FUNCTION_BLOCK BLOCK_POMP_1E_PCR_PPM_ASS_ETHERCAT

(* Historique des versions*)
(* VERSION 1.0 - 05/2015 - GV - affaire 9070*)
(* VERSION 2.0 - 10/2022 - GV - ajout gestion roots *)


(* BLOCK GESTION POMPAGE CRYO ON BOARD ENCEINTE *)
(*	Gestion pompage enceinte sans sas constitué de :
	Pompe primaire pour prévidage, regen cryo et pompage interjoint
	Pompe cryogénique on-board CTI pour le pompage secondaire
	Vanne de pompage primaire enceinte
	Vanne de remise à atmosphère enceinte
	Vanne de pompage inter-joint (optionnelle)
	Vanne secondaire asservie, pilotée par ethercatf
*)

VAR_INPUT
(*information générale*)
	RESET:					BOOL;
	MANUAL:					BOOL;
	CTRL_PLC:				BOOL;
	I_Prep_Ventil_Ok:		BOOL;		(*information externe indiquant que l'enceinte est prête à être ventilée par ex. circulation d'eau à l'arrêt
										ou polycold arreté ou basculement en eau chaude ok ...*)
	I_Fin_Ventil:			BOOL;		(*information externe de fin de ventilation de l'enceinte  *)
	I_Stop_Mesure_OK:		BOOL;		(*information externe indiquant que les jauges ont été stoppées prélablement à la ventilation de l'enceinte*)
	IN_Pressure_RP:			REAL;		(*interfaçage avec M11.state_pression du PRG correspondant*)
	I_Ref_OK:				BOOL;		(*information externe indiquant que le refroidissement est ok pour démarrer les pompes*)
	
(*Gestion régen partielle*)
	IN_Temp_Etage1:			REAL;
	PRM_Temp_Post_Purge:	REAL;
	PRM_Tim_Post_Purge:		TIME;

(*Paramètres et commandes du test de remontée de pression*)
	PRM_Pr_test:			REAL;		(*Pression initiale de test de remontée*)
	PRM_Tim_test:			TIME;		(*Durée d'attente en test*)
	CO_Stop_Test_RP:		BOOL;		(*Demande arrêt test remontée de pression*)

(*sécurité*)
	IN_FE11T:				BOOL;		(*indicateur enceinte fermée - capteur 1*)
	IN_FE12T:				BOOL;		(*indicateur enceinte fermée - capteur 2*)
	IN_VT11F:				BOOL;		(*clapet SAS enceinte fermé*)

(*seuil de vide*)
	TH_Vide_Primaire:		BOOL;		(*Pression enceinte <= Seuil de fin de pompage primaire*)
	TH_Grosse_Fuite:		BOOL;		(*Pression enceinte <= Seuil de detection de grosse fuite enceinte*)
	TH_Atm:					BOOL;		(*pression enceinte >= Seuil pression atm. de fin de ventilation*)
	TH_RP_Enc:				BOOL;		(*pression enceinte <= Pression max. dans l'enceinte*)
	TH_Test_RP:				BOOL;		(*Pression <= Seuil de pression de test*)

(*composant de la fonction*)
	VP11:					BLOCK_ACTUATOR;									(*vanne de pompage primaire enceinte *)
	VH11:					BLOCK_ACTUATOR;									(*vanne de ventilation de l'enceinte*)
	PP11:					BLOCK_PPM;										(*Pompe primaire enceinte*)
	PR11:					BLOCK_PPM;										(*Pompe roots enceinte*)
	PS11:					BLOCK_PCR_CTI_OB;								(*Pompe cryogénique on board  enceinte*)
	VS11:					BLOCK_VVAT_653_ETHERCAT;						(*Vanne secondaire asservie pompage enceinte*)
	VINT:					BLOCK_ACTUATOR;									(*Vanne de pompage dans les interjoints*)

(*défaut*)
	DEF_PPrim:				PRCDEF;										(*défaut temps de pompage primaire dans l'enceinte*)
	DEF_Vent:				PRCDEF;										(*défaut temps de ventilation enceinte*)
	DEF_RP_enc:				PRCDEF;	 									(*défaut perte seuil de pompage primaire en pompage secondaire*)
	DEF_TGF:				PRCDEF;										(*défaut détection trés grosse fuite*)

(*opération*)
	OP_Marche_Pompes:			BLOCK_OPERATION;								(*opération marche pompe*)
	OP_Arret_Pompes:			BLOCK_OPERATION;								(*opération arrêt pompe*)
	OP_Isolement:				BLOCK_OPERATION;								(*opération stand-by*)
	OP_Ventilation:				BLOCK_OPERATION;								(*opération ventilation*)
	OP_Pompage_Sec:				BLOCK_OPERATION;								(*opération pompage secondaire*)
	OP_Pompage_Prim:			BLOCK_OPERATION;								(*opération pompage primaire*)
	OP_Pompage_Proc:			BLOCK_OPERATION;								(*opération pompage en procédé*)
	OP_Purge:					BLOCK_OPERATION;								(*opération purge*)
	OP_Regen:					BLOCK_OPERATION;								(*opération régénération pompe cryogénique*)
	OP_Regen_Part:				BLOCK_OPERATION;								(*opération de régénération partielle pompe cryogénique*)
	OP_Test_RP:					BLOCK_OPERATION;								(*opération test RP*)
	G7_pompage_interjoint:		BLOCK_G7;

END_VAR

VAR_INPUT PERSISTENT
(*paramètre*)
	PRM_Tim_SurVentil_E:		TIME;	(*durée du temps de surventilation*)
	PRM_Tim_Purge:				TIME;	(*durée du maintien pompage primaire en purge*)
	PRM_Tim_Arret_PP11:			TIME;	(*durée avant arrêt de la pompe primaire*)
	PRM_Pr_Atm:					REAL;	(*Pression atmosphérique dans l'enceinte*)
	PRM_Pr_PPrim:				REAL;	(*Pression de fin de pompage primaire dans l'enceinte*)
	PRM_Pr_RP_PPrim:			REAL;	(*Pression max admissible dans l'enceinte en pompage secondaire dans l'enceinte*)
	PRM_Pr_TGF:					REAL;	(*Pression de détection trés grosse fuite dans l'enceinte*)
	PRM_N_Purge:				USINT;	(*Nombre de cycles de purge pompage/ventilation*)
	CONF_Pompage_interjoint:	BOOL;	(*Utilisation de la pompe primaire pour le pompage interjoint sur l'enceinte*)
	CONF_VINT:					BOOL;	(*Utilisation d'une vanne d'isolement sur le pompage interjoint*)
	CONF_Volume_Enceinte:		REAL;	(*Volume pour RP*)

	PRM_Tim_Prep_Ventil:		TIME;	(*temporisation de prép ventilation (eau chaude suffisemment longtemps) *)

	(*Entité*)
	IsAssembly:		BOOL;		(*entité : ensemble*)
	IdXML:			STRING;		(*nom entité : identifiant pour recherche dans dico*)
	TagXML:			UINT;		(*nom entité : identifiant pour recherche dans dico*)
	IdParent:		STRING;		(*MNEMO de l'appelant*)
	MNEMO:			STRING;		(*MNEMO de l'entité*)
END_VAR


VAR_OUTPUT
	RQ_Prep_Ventil_Enc:		BOOL;											(*demande de préparation avant ventilation (réchauffement, arrêt eau ....*)
	RQ_Stop_Mesure_Enc:		BOOL;											(*demande d'arrêt de la mesure avant ventilation - Les blocs jauges concernés utilise
																			cette information pour stoppée les jauges préalablement à la ventilation*)
END_VAR

VAR_IN_OUT
END_VAR

VAR
	VAR_Reset_Sortie:					BOOL;
	TIMER_SurVentilation_Enc:			TON;		(*Temporistion de surventilation enceinte*)
	TIMER_Purge:						TON;		(*Temporisation de maintien pompage primaire en purge*)
	TIMER_Pompage_Interjoint:			TON;		(*Temporisation d'ouverture de la vanne de pompage interjoint*)
	TIMER_Arret_Roots:					TON;		(*Temporisation arrêt roots après prévidage*)
	TIMER_Arret_PP11:					TON;		(*Temporisation arrêt pompe primaire*)
	VAR_mem_isolement:					BOOL;
	VAR_Iter_Purge:						USINT;

	(*Pour RP*)
	VAR_Mem_Pression_Deb:		REAL;
	VAR_Mem_Pression_Fin:		REAL;
	VAR_Indicateur_Test:		REAL; 		(*résultat final*)
	TIMER_attente_test:			TON;		(*Temporisation pour test de remontée en pression*)
	FM_etape4:					R_TRIG;

	(*Pour prep ventil*)
	TIM_Prep_ventil:			TON;		(*timer de préparation ventil*)

	(*Pour regen*)
	FM_REGEN:						R_TRIG;		(* FM pompe cryogénique en régénération*)
	FD_REGEN:						F_TRIG;		(* FD pompe cryogénique en régénération*)
	TIMER_Post_Purge:				TON;		(*tempo max attente de retombée température après purge en regen partielle*)
	TIMER_etape6_regen:				TON;
END_VAR

PRL();

(*appel des opérations*)
ACT_ARRET_POMPES();
ACT_ISOLEMENT();
ACT_MARCHE_POMPES();
ACT_POMPAGE_PRIM();
ACT_POMPAGE_PROC();
ACT_POMPAGE_SEC();
ACT_VENTILATION();
ACT_PURGE();
ACT_REGEN();
ACT_REGEN_PART();
ACT_TEST_RP();
ACT_POMPAGE_INTERJOINT();

(*action en sortie*)
POST();

ACTION ACT_ARRET_POMPES:
(* OPERATION ARRET POMPES*)
(* arrêt des pompes*)

(*initialisation de l'opération*)
OP_ARRET_POMPES(
	CTRL_PLC:= CTRL_PLC,
	RESET:= RESET,
	ENABLE_INT:=TRUE,
	MANUAL:= MANUAL,
	ON_AUTO_INT:= (PP11.STATE_NOK AND PR11.STATE_NOK) AND (NOT OP_Pompage_Prim.Etape.0 OR NOT OP_Purge.Etape.0),
	RESTART_ENABLE_IF_OK:= FALSE,
	N_STEP_OP_OK:= 5,
	N_STEP_OP_NOK:=0);

(*appel de l'action de préparation de l'opération*)
OP_ARRET_POMPES.PRL();


(*GRAFCET*)
(* initialisation du grafcet*)
IF 		OP_Arret_Pompes.ETAPE = 0 THEN
				OP_Arret_Pompes.ETAPE.0 := TRUE;
(*repositionnement sur étape 0*)
ELSIF	MANUAL OR RESET OR OP_Marche_Pompes.ETAPE.1 THEN
				OP_Arret_Pompes.ETAPE := 0;			(*RAZ grafcet*)
				OP_Arret_Pompes.ETAPE.0:=TRUE;
(*étape 0-1*)
ELSIF 	OP_Arret_Pompes.ETAPE.0
		AND OP_Arret_Pompes.MARCHE_OP THEN
				OP_Arret_Pompes.ETAPE.1:=TRUE;
				OP_Arret_Pompes.ETAPE.0:=FALSE;
(*étape 1-2*)
ELSIF	OP_Arret_Pompes.ETAPE.1
		AND OP_Marche_Pompes.ETAPE.0  THEN
				OP_Arret_Pompes.Etape.2:=TRUE;
				OP_Arret_Pompes.Etape.1:=FALSE;
(*étape 2-3*)
ELSIF 	OP_Arret_Pompes.Etape.2
		AND (OP_Isolement.OK OR VAR_mem_isolement)
		AND (VINT.STATE_Off OR NOT CONF_VINT)
		 THEN
				OP_Arret_Pompes.Etape.3:=TRUE;
				OP_Arret_Pompes.Etape.2:=FALSE;
(*étape 3-4*)
ELSIF 	OP_Arret_Pompes.Etape.3
		AND	Timer_Arret_PP11.Q THEN 
				OP_Arret_Pompes.Etape.4:=TRUE;
				OP_Arret_Pompes.Etape.3:=FALSE;
(*étape 4-5*)
ELSIF	OP_Arret_Pompes.Etape.4
		AND PP11.STATE_Off AND PR11.STATE_Off AND PS11.STATE_Ar THEN
				OP_Arret_Pompes.Etape.5:=TRUE;
				OP_Arret_Pompes.Etape.4:=FALSE;
END_IF;

(*cloture du traitement de l'opération*)
OP_Arret_Pompes.POST();

(************************************************************************)
(*Gestion de la mémoire de la demande d'isolement de l'enceinte*)
(************************************************************************)
IF 		OP_Ventilation.Etape.9 THEN
	VAR_mem_isolement	:=	TRUE;
ELSIF	NOT OP_Pompage_Prim.AR OR NOT OP_Pompage_Sec.AR OR NOT OP_Pompage_Proc.AR OR NOT OP_Purge.AR THEN
	VAR_mem_isolement	:=	FALSE;
END_IF
(*IF OP_Arret_pompes.Etape.2 AND (NOT OP_Pompage_Prim.Etape.0  OR NOT OP_Pompage_Proc.Etape.0 OR NOT OP_Pompage_Sec.Etape.0) THEN
	VAR_mem_isolement_enceinte := TRUE;
END_IF;
IF OP_Arret_pompes.Etape.0 OR OP_Arret_Pompes.Etape.3 THEN
	VAR_mem_isolement_enceinte := FALSE;
END_IF;*)
END_ACTION

ACTION ACT_ISOLEMENT:
(*OPERATION ISOLEMENT ENCEINTE*)
(*isolement de l'enceinte*)

(*initialisation de l'opération*)
OP_Isolement(
	CTRL_PLC:= CTRL_PLC,
	RESET:= RESET,
	ENABLE_INT:=TRUE,
	MANUAL:= MANUAL,
	ON_AUTO_INT:= 	((DEF_TGF.DEF OR DEF_RP_enc.DEF) AND (NOT OP_Pompage_Prim.Etape.0 OR NOT OP_Pompage_Sec.Etape.0 OR NOT OP_Pompage_proc.Etape.0))
					OR (PS11.STATE_Nok AND (NOT OP_Pompage_Sec.Etape.0 OR NOT OP_Pompage_proc.Etape.0))
					OR (PP11.STATE_Nok AND NOT OP_Pompage_Prim.Etape.0)
					OR (PR11.STATE_NOK AND NOT OP_Pompage_Prim.Etape.0),
	RESTART_ENABLE_IF_OK:= FALSE,
	N_STEP_OP_OK:= 4,
	N_STEP_OP_NOK:=0);

(*appel de l'action de préparation de l'opération*)
OP_Isolement.PRL();


(*GRAFCET*)
(* initialisation du grafcet*)
IF 		OP_Isolement.Etape = 0
		THEN
				OP_Isolement.Etape.0	:= TRUE;
(*repositionnement sur étape 0*)
ELSIF	MANUAL OR RESET OR OP_pompage_sec.Etape.1 OR OP_Pompage_Proc.Etape.1 OR Op_Pompage_Prim.Etape.1
		OR OP_ventilation.Etape.2 OR OP_Ventilation.Etape.9 OR OP_Purge.Etape.1 THEN
				OP_Isolement.Etape := 0;
				OP_Isolement.Etape.0:=TRUE;
(*étape 0-1*)
ELSIF 	OP_Isolement.Etape.0
		AND(
		OP_Isolement.Marche_OP OR
		OP_ventilation.Etape.1 OR
		OP_Test_RP.Etape.3 OR
		(OP_Arret_Pompes.Etape.2 AND NOT VAR_mem_isolement) OR
		OP_Regen.Etape.2 OR OP_Regen_Part.Etape.2
		)
		THEN
				OP_Isolement.Etape.1:=TRUE;
				OP_Isolement.Etape.0:=FALSE;
(*étape 1-2*)
ELSIF	OP_Isolement.Etape.1
		AND OP_Pompage_Proc.Etape.0
		AND OP_Pompage_Prim.Etape.0
		AND OP_Pompage_Sec.Etape.0
		AND (OP_Ventilation.Etape.0 OR OP_Ventilation.Etape.1)
		AND (OP_Purge.Etape.0 OR (OP_Purge.Etape.4 AND OP_Ventilation.Etape.1))
		THEN
				OP_Isolement.Etape.2:=TRUE;
				OP_Isolement.Etape.1:=FALSE;
(*étape 2-3*)
ELSIF 	OP_Isolement.Etape.2 AND
		VP11.STATE_Off AND
		VS11.STATE_Off AND
		VH11.STATE_Off  THEN
				OP_Isolement.Etape.3:=TRUE;
				OP_Isolement.Etape.2:=FALSE;
(*étape 3-4*)
ELSIF	OP_Isolement.Etape.3
		AND ((PP11.STATE_Off AND PR11.STATE_Off) OR PS11.STATE_Regen OR CONF_Pompage_interjoint) THEN
				OP_isolement.Etape.4:=TRUE;
				OP_isolement.Etape.3:=FALSE;
END_IF;

(*cloture du traitement de l'opération*)
OP_Isolement.POST();
END_ACTION

ACTION ACT_MARCHE_POMPES:
(* OPERATION MARCHE POMPES*)
(* mise en marche des pompes*)

(*initialisation de l'opération*)
OP_MARCHE_POMPES(
	CTRL_PLC:= CTRL_PLC,
	RESET:= RESET,
	ENABLE_INT:=TRUE,
	MANUAL:= MANUAL,
	ON_AUTO_INT:= TRUE,
	RESTART_ENABLE_IF_OK:= FALSE,
	N_STEP_OP_OK:= 5,
	N_STEP_OP_NOK:=0);

(*appel de l'action de préparation de l'opération*)
OP_MARCHE_POMPES.PRL();


(*GRAFCET*)
(* initialisation du grafcet*)
IF 		OP_MARCHE_POMPES.ETAPE = 0
		THEN
				OP_MARCHE_POMPES.ETAPE.0 := TRUE;
(*repositionnement sur étape 0*)
ELSIF	MANUAL OR RESET OR OP_ARRET_POMPES.ETAPE.1
		THEN
				OP_MARCHE_POMPES.ETAPE := 0;			(*RAZ grafcet*)
				OP_MARCHE_POMPES.ETAPE.0:=TRUE;
(*étape 0-1*)
ELSIF 	OP_MARCHE_POMPES.ETAPE.0
		AND (OP_MARCHE_POMPES.MARCHE_OP OR OP_POMPAGE_SEC.ETAPE.2
			OR (OP_Regen.Etape.5 AND TH_Atm))
		THEN
				OP_MARCHE_POMPES.ETAPE.1:=TRUE;
				OP_MARCHE_POMPES.ETAPE.0:=FALSE;
(*étape 1-2*)
ELSIF	OP_MARCHE_POMPES.ETAPE.1
		AND OP_ARRET_POMPES.ETAPE.0 AND PR11.STATE_Off AND I_Ref_Ok
		THEN
				OP_MARCHE_POMPES.ETAPE.2:=TRUE;
				OP_MARCHE_POMPES.ETAPE.1:=FALSE;
(*étape 2-3*)
ELSIF 	OP_MARCHE_POMPES.ETAPE.2
		AND (PP11.STATE_On OR NOT CONF_Pompage_interjoint)
		THEN
				OP_MARCHE_POMPES.ETAPE.3:=TRUE;
				OP_MARCHE_POMPES.ETAPE.2:=FALSE;
(*étape 3-4*)
ELSIF	OP_MARCHE_POMPES.ETAPE.3
		THEN
				OP_MARCHE_POMPES.ETAPE.4:=TRUE;
				OP_MARCHE_POMPES.ETAPE.3:=FALSE;
(*étape 4-5*)
ELSIF 	OP_MARCHE_POMPES.ETAPE.4
		AND PS11.STATE_On AND PS11.STATE_Ok AND NOT PS11.STATE_Regen
		THEN
				OP_MARCHE_POMPES.ETAPE.5:=TRUE;
				OP_MARCHE_POMPES.ETAPE.4:=FALSE;
(*étape 5-4*)
ELSIF 	OP_MARCHE_POMPES.ETAPE.5
		AND (PS11.STATE_Regen OR NOT PS11.STATE_Ok)		THEN
				OP_MARCHE_POMPES.ETAPE.4:=TRUE;
				OP_MARCHE_POMPES.ETAPE.5:=FALSE;
END_IF;

(*cloture du traitement de l'opération*)
OP_MARCHE_POMPES.POST();
END_ACTION

ACTION ACT_POMPAGE_INTERJOINT:
(*GRAFCET*)
(* initialisation du grafcet*)
IF 		G7_pompage_interjoint.etape = 0
		THEN
				G7_pompage_interjoint.etape.0 := TRUE;
(*repositionnement sur étape 0*)
ELSIF	MANUAL OR RESET
		OR (NOT OP_POMPAGE_SEC.OK AND NOT OP_Pompage_Proc.OK AND NOT OP_Pompage_Proc.EC)
		OR NOT CONF_Pompage_interjoint OR NOT CONF_VINT
		THEN
				G7_pompage_interjoint.etape := 0;			(*RAZ grafcet*)
				G7_pompage_interjoint.etape.0:=TRUE;
(*étape 0-1*)
ELSIF 	G7_pompage_interjoint.etape.0
		AND (OP_POMPAGE_SEC.OK OR OP_Pompage_Proc.EC OR OP_Pompage_Proc.OK)
		THEN
				G7_pompage_interjoint.etape.1:=TRUE;
				G7_pompage_interjoint.etape.0:=FALSE;
(*étape 1-2*)
ELSIF	G7_pompage_interjoint.etape.1
		AND TIMER_pompage_interjoint.Q
		THEN
				G7_pompage_interjoint.etape.2:=TRUE;
				G7_pompage_interjoint.etape.1:=FALSE;
END_IF;

G7_pompage_interjoint.POST();
END_ACTION

ACTION ACT_POMPAGE_PRIM:
(*OPERATION POMPAGE PRIMAIRE ENCEINTE*)
(*pompage primaire dans l'enceinte*)

(*initialisation de l'opération*)
OP_POMPAGE_PRIM(
	CTRL_PLC:= CTRL_PLC,
	RESET:= RESET,
	ENABLE_INT:= OP_Purge.Etape.0 AND IN_FE11T AND IN_FE12T,
	MANUAL:= MANUAL,
	RESTART_ENABLE_IF_OK:= FALSE,
	N_STEP_OP_OK:= 5,
	N_STEP_OP_NOK:=0);

(*appel de l'action de préparation de l'opération*)
OP_POMPAGE_PRIM.PRL();


(*GRAFCET*)
(* initialisation du grafcet*)
IF 		OP_Pompage_Prim.Etape = 0
		THEN
				OP_Pompage_Prim.Etape.0:= TRUE;
(*repositionnement sur étape 0*)
ELSIF	MANUAL OR RESET OR OP_Isolement.Etape.1 OR OP_Pompage_Sec.Etape.4
		OR OP_Pompage_Proc.Etape.1
		THEN
				OP_Pompage_Prim.ETAPE := 0;
				OP_Pompage_Prim.Etape.0:=TRUE;
(*étape 0-1*)
ELSIF 	OP_Pompage_Prim.Etape.0
		AND (OP_Pompage_Prim.Marche_OP OR OP_Pompage_Sec.Etape.3 OR OP_Purge.Etape.2)
		THEN
				OP_Pompage_Prim.Etape.1:=TRUE;
				OP_Pompage_Prim.Etape.0:=FALSE;
(*étape 1-2*)
ELSIF	OP_Pompage_Prim.Etape.1
		AND OP_Isolement.Etape.0
		AND OP_Ventilation.Etape.0
		AND OP_Pompage_Proc.Etape.0
		AND (OP_Pompage_Sec.Etape.0 OR OP_Pompage_Sec.Etape.3)
		AND (OP_Purge.Etape.0 OR OP_Purge.Etape.6 OR OP_Purge.Etape.2)
		AND VS11.STATE_Off
		AND VH11.STATE_Off
		THEN
				OP_Pompage_Prim.Etape.2:=TRUE;
				OP_Pompage_Prim.Etape.1:=FALSE;

(*étape 2-3*)
ELSIF 	OP_Pompage_prim.Etape.2
		THEN
				OP_Pompage_Prim.Etape.3:=TRUE;
				OP_Pompage_Prim.Etape.2:=FALSE;
(*étape 3-4*)
ELSIF	OP_Pompage_Prim.Etape.3
		AND PP11.STATE_On AND PR11.STATE_On THEN
				OP_Pompage_Prim.Etape.4:=TRUE;
				OP_Pompage_Prim.Etape.3:=FALSE;
(*étape 4-5*)
ELSIF 	OP_Pompage_Prim.Etape.4
		AND VP11.STATE_On
		THEN
				OP_Pompage_Prim.Etape.5:=TRUE;
				OP_Pompage_Prim.Etape.4:=FALSE;
END_IF;

(*cloture du traitement de l'opération*)
OP_Pompage_Prim.POST();
END_ACTION

ACTION ACT_POMPAGE_PROC:
(*OPERATION POMPAGE PROCEDE*)
(*pompage procede dans l'enceinte*)

(*initialisation de l'opération*)
OP_Pompage_Proc(
	CTRL_PLC:= CTRL_PLC,
	RESET:= RESET,
	ENABLE_INT:= OP_POMPAGE_SEC.OK OR OP_Pompage_Proc.OK,
	MANUAL:= MANUAL,
	RESTART_ENABLE_IF_OK:= FALSE,
	N_STEP_OP_OK:= 3,
	N_STEP_OP_NOK:=0);

(*appel de l'action de préparation de l'opération*)
OP_Pompage_Proc.PRL();


(*GRAFCET*)
(* initialisation du grafcet*)
IF 		OP_Pompage_Proc.Etape = 0
		THEN
				OP_Pompage_Proc.Etape.0:= TRUE;
(*repositionnement sur étape 0*)
ELSIF	MANUAL OR RESET OR OP_Isolement.Etape.1 OR OP_Pompage_Prim.Etape.1 OR OP_Pompage_Sec.Etape.1
		OR OP_Purge.Etape.1
		THEN
				OP_Pompage_Proc.Etape := 0;
				OP_Pompage_Proc.Etape.0:=TRUE;
(*étape 0-1*)
ELSIF 	OP_Pompage_Proc.Etape.0
		AND OP_Pompage_Proc.Marche_OP
		THEN
				OP_Pompage_Proc.Etape.1:=TRUE;
				OP_Pompage_Proc.Etape.0:=FALSE;
(*étape 1-2*)
ELSIF	OP_Pompage_Proc.Etape.1
		AND OP_Pompage_Sec.Etape.0
		THEN
				OP_Pompage_Proc.Etape.2:=TRUE;
				OP_Pompage_Proc.Etape.1:=FALSE;
(*étape 2-3*)
ELSIF 	OP_Pompage_proc.Etape.2
		AND VS11.STATE_Lam THEN
				OP_Pompage_Proc.Etape.3:=TRUE;
				OP_Pompage_Proc.Etape.2:=FALSE;
(*étape 3-2*)
ELSIF 	OP_Pompage_Proc.Etape.3
		AND OP_Pompage_Proc.Marche_OP
		THEN
				OP_Pompage_Proc.Etape.2:=TRUE;
				OP_Pompage_Proc.Etape.3:=FALSE;
END_IF;

(*cloture du traitement de l'opération*)
OP_Pompage_Proc.POST();
END_ACTION

ACTION ACT_POMPAGE_SEC:
(*OPERATION POMPAGE SECONDAIRE ENCEINTE*)
(*pompage secondaire dans l'enceinte*)

(*initialisation de l'opération*)
OP_pompage_sec(
	CTRL_PLC:= CTRL_PLC,
	RESET:= RESET,
	ENABLE_INT:=IN_FE11T AND IN_FE12T AND NOT PS11.STATE_Regen,
	MANUAL:= MANUAL,
	RESTART_ENABLE_IF_OK:= FALSE,
	N_STEP_OP_OK:= 7,
	N_STEP_OP_NOK:=0);

(*appel de l'action de préparation de l'opération*)
OP_Pompage_Sec.PRL();


(*GRAFCET*)
(* initialisation du grafcet*)
IF 		OP_Pompage_Sec.Etape = 0
		THEN
				OP_Pompage_Sec.Etape.0:= TRUE;
(*repositionnement sur étape 0*)
ELSIF	MANUAL OR RESET OR OP_Isolement.Etape.1 OR OP_Pompage_Proc.Etape.1
		OR (OP_Pompage_Prim.Etape.1 AND NOT OP_Pompage_Sec.Etape.3) OR OP_Purge.Etape.1
		THEN
				OP_Pompage_Sec.Etape := 0;
				OP_Pompage_Sec.Etape.0:=TRUE;
(*étape 0-1*)
ELSIF 	OP_Pompage_Sec.Etape.0 AND
		(OP_Pompage_Sec.Marche_OP OR OP_Purge.Etape.6 OR
			OP_Test_RP.Etape.2 OR OP_Test_RP.Etape.7
		OR (OP_Regen.Etape.5 AND NOT TH_Atm AND OP_Pompage_Sec.ENABLE_INT))
		THEN
				OP_Pompage_Sec.Etape.1:=TRUE;
				OP_Pompage_Sec.Etape.0:=FALSE;
(*étape 1-2*)
ELSIF	OP_Pompage_Sec.Etape.1
		AND OP_Isolement.Etape.0
		AND OP_Ventilation.Etape.0
		AND OP_Pompage_Proc.Etape.0
		AND (OP_Purge.Etape.0 OR OP_Purge.Etape.6)
		THEN
				OP_Pompage_Sec.Etape.2:=TRUE;
				OP_Pompage_Sec.Etape.1:=FALSE;
(*étape 2-3*)
ELSIF 	OP_Pompage_Sec.Etape.2
		AND OP_MARCHE_POMPES.ok AND NOT TH_Vide_Primaire AND VH11.STATE_Off
		THEN
				OP_Pompage_Sec.Etape.3:=TRUE;
				OP_Pompage_Sec.Etape.2:=FALSE;
(*étape 2-4*)
ELSIF 	OP_Pompage_Sec.Etape.2
		AND OP_MARCHE_POMPES.ok AND TH_Vide_Primaire AND VH11.STATE_Off
		THEN
				OP_Pompage_Sec.Etape.4:=TRUE;
				OP_Pompage_Sec.Etape.2:=FALSE;
(*étape 3-4*)
ELSIF	OP_Pompage_Sec.Etape.3
		AND	OP_POMPAGE_PRIM.ok  AND TH_Vide_Primaire
		THEN
				OP_Pompage_Sec.Etape.4:=TRUE;
				OP_Pompage_Sec.Etape.3:=FALSE;
(*étape 4-5*)
ELSIF	OP_Pompage_Sec.Etape.4
		AND VP11.STATE_Off
		AND  OP_POMPAGE_PRIM.AR   THEN
				OP_Pompage_Sec.Etape.5:=TRUE;
				OP_Pompage_Sec.Etape.4:=FALSE;
(*étape 5-6*)
ELSIF 	OP_Pompage_Sec.Etape.5
		AND (PP11.STATE_Off AND PR11.STATE_Off OR CONF_Pompage_interjoint)
		THEN
				OP_Pompage_Sec.Etape.6:=TRUE;
				OP_Pompage_Sec.Etape.5:=FALSE;
(*étape 6-7*)
ELSIF 	OP_Pompage_Sec.Etape.6
		AND VS11.STATE_On
		THEN
				OP_Pompage_Sec.Etape.7:=TRUE;
				OP_Pompage_Sec.Etape.6:=FALSE;
END_IF;

(*cloture du traitement de l'opération*)
OP_Pompage_Sec.POST();
END_ACTION

ACTION ACT_PURGE:
(*OPERATION PURGE*)
(*purge enceinte : pompage primaire pendant un temps donné puis ventilation, répété X fois*)

(*initialisation de l'opération*)
OP_Purge(
	CTRL_PLC:= CTRL_PLC,
	RESET:= RESET,
	ENABLE_INT:= IN_FE11T AND IN_FE12T AND OP_Test_RP.AR,
	MANUAL:= MANUAL,
	RESTART_ENABLE_IF_OK:= FALSE,
	N_STEP_OP_OK:= 7,
	N_STEP_OP_NOK:=0);

(*appel de l'action de préparation de l'opération*)
OP_Purge.PRL();


(*GRAFCET*)
(* initialisation du grafcet*)
IF 		OP_Purge.Etape = 0
		THEN
				OP_Purge.Etape.0:= TRUE;
(*repositionnement sur étape 0*)
ELSIF	MANUAL OR RESET OR OP_Arret_Pompes.Etape.1
		OR (OP_Isolement.Etape.1 AND NOT OP_Ventilation.Etape.1)
		OR (OP_Pompage_Sec.Etape.1 AND NOT OP_Purge.Etape.6)
		THEN
				OP_Purge.Etape := 0;
				OP_Purge.Etape.0:=TRUE;
(*étape 0-1*)
ELSIF 	OP_Purge.Etape.0
		AND OP_Purge.Marche_OP
		THEN
				OP_Purge.Etape.1:=TRUE;
				OP_Purge.Etape.0:=FALSE;
(*étape 1-2*)
ELSIF	OP_Purge.Etape.1
		AND OP_Pompage_Sec.Etape.0 AND OP_Pompage_Prim.Etape.0 AND OP_Pompage_Proc.Etape.0
		AND OP_Ventilation.Etape.0 AND OP_Isolement.Etape.0
		THEN
				OP_Purge.Etape.2:=TRUE;
				OP_Purge.Etape.1:=FALSE;
(*étape 2-3*)
ELSIF 	OP_Purge.Etape.2
		AND OP_Pompage_Prim.OK AND TH_Vide_Primaire
		THEN
				OP_Purge.Etape.3:=TRUE;
				OP_Purge.Etape.2:=FALSE;
(*étape 3-4*)
ELSIF 	OP_Purge.Etape.3
		AND TIMER_Purge.Q
		THEN
				OP_Purge.Etape.4:=TRUE;
				OP_Purge.Etape.3:=FALSE;
(*étape 3-2*)
ELSIF 	OP_Purge.Etape.3
		AND NOT OP_Pompage_Prim.OK
		THEN
				OP_Purge.Etape.2:=TRUE;
				OP_Purge.Etape.3:=FALSE;
(*étape 4-5*)
ELSIF 	OP_Purge.Etape.4
		AND TH_Atm
		THEN
				OP_Purge.Etape.5:=TRUE;
				OP_Purge.Etape.4:=FALSE;
(*étape 5-2*)
ELSIF 	OP_Purge.Etape.5
		AND (VAR_Iter_Purge < PRM_N_Purge)
		THEN
				OP_Purge.Etape.2:=TRUE;
				OP_Purge.Etape.5:=FALSE;
(*étape 5-6*)
ELSIF 	OP_Purge.Etape.5
		AND (VAR_Iter_Purge >= PRM_N_Purge)
		THEN
				OP_Purge.Etape.6:=TRUE;
				OP_Purge.Etape.5:=FALSE;
(*étape 6-7*)
ELSIF 	OP_Purge.Etape.6
		AND OP_Pompage_Sec.EC
		THEN
				OP_Purge.Etape.7:=TRUE;
				OP_Purge.Etape.6:=FALSE;
END_IF;

(*cloture du traitement de l'opération*)
OP_Purge.POST();
END_ACTION

ACTION ACT_REGEN:
(*OPERATION REGENERATION POMPE CRYOGENIQUE*)
(*isolement pompage et lancement régénération*)

(*initialisation de l'opération*)
OP_Regen(
	CTRL_PLC:= CTRL_PLC,
	RESET:= RESET,
	ENABLE_INT:= OP_Test_RP.AR AND NOT OP_Marche_Pompes.AR,
	MANUAL:= MANUAL,
	RESTART_ENABLE_IF_OK:= FALSE,
	N_STEP_OP_OK:= 6,
	N_STEP_OP_NOK:=0);

(*appel de l'action de préparation de l'opération*)
OP_Regen.PRL();


(*GRAFCET*)
(* initialisation du grafcet*)
IF 		OP_Regen.Etape = 0
		THEN
				OP_Regen.Etape.0:= TRUE;
(*repositionnement sur étape 0*)
ELSIF	MANUAL OR RESET OR OP_Arret_Pompes.Etape.1
		THEN
				OP_Regen.Etape := 0;
				OP_Regen.Etape.0:=TRUE;
(*étape 0-1*)
ELSIF 	OP_Regen.Etape.0
		AND (OP_Regen.Marche_OP OR (FM_REGEN.Q AND NOT MANUAL AND NOT OP_Regen_Part.EC))
		THEN
				OP_Regen.Etape.1:=TRUE;
				OP_Regen.Etape.0:=FALSE;
(*étape 1-2*)
ELSIF	OP_Regen.Etape.1
		THEN
				OP_Regen.Etape.2:=TRUE;
				OP_Regen.Etape.1:=FALSE;
(*étape 2-3*)
ELSIF 	OP_Regen.Etape.2
		AND (OP_Isolement.Etape.4 OR (OP_Pompage_Prim.Etape.0 AND OP_Pompage_Proc.Etape.0 OR OP_Pompage_Sec.Etape.0 OR OP_Purge.Etape.0))
		THEN
				OP_Regen.Etape.3:=TRUE;
				OP_Regen.Etape.2:=FALSE;
(*étape 3-4*)
ELSIF	OP_Regen.Etape.3 AND PS11.STATE_Regen
		THEN
				OP_Regen.Etape.4:=TRUE;
				OP_Regen.Etape.3:=FALSE;
(*étape 4-5*)
ELSIF	OP_Regen.Etape.4 AND NOT PS11.STATE_Regen
		THEN
				OP_Regen.Etape.5:=TRUE;
				OP_Regen.Etape.4:=FALSE;
(*étape 5-6*)
ELSIF	OP_Regen.Etape.5
		AND (OP_Pompage_Sec.OK OR (OP_Marche_Pompes.OK AND (TH_Atm OR NOT OP_Pompage_Sec.ENABLE_INT)))
		THEN
				OP_Regen.Etape.6:=TRUE;
				OP_Regen.Etape.5:=FALSE;
(*étape 6-0*)
ELSIF	OP_Regen.Etape.6
		AND TIMER_etape6_regen.Q
		THEN
				OP_Regen.Etape.0:=TRUE;
				OP_Regen.Etape.6:=FALSE;
END_IF;

(*cloture du traitement de l'opération*)
OP_Regen.POST();
END_ACTION

ACTION ACT_REGEN_PART:
(*OPERATION REGENERATION POMPE CRYOGENIQUE*)
(*isolement pompage et lancement régénération*)

(*initialisation de l'opération*)
OP_Regen_Part(
	CTRL_PLC:= CTRL_PLC,
	RESET:= RESET,
	ENABLE_INT:= OP_Test_RP.AR AND NOT OP_Marche_Pompes.AR,
	MANUAL:= MANUAL,
	RESTART_ENABLE_IF_OK:= FALSE,
	N_STEP_OP_OK:= 6,
	N_STEP_OP_NOK:=0);

(*appel de l'action de préparation de l'opération*)
OP_Regen_Part.PRL();


(*GRAFCET*)
(* initialisation du grafcet*)
IF 		OP_Regen_Part.Etape = 0
		THEN
				OP_Regen_Part.Etape.0:= TRUE;
(*repositionnement sur étape 0*)
ELSIF	MANUAL OR RESET OR OP_Arret_Pompes.Etape.1
		OR OP_Pompage_Sec.Etape.1 OR OP_Pompage_Prim.Etape.1
		THEN
				OP_Regen_Part.Etape := 0;
				OP_Regen_Part.Etape.0:=TRUE;
(*étape 0-1*)
ELSIF 	OP_Regen_Part.Etape.0
		AND OP_Regen_Part.Marche_OP
		THEN
				OP_Regen_Part.Etape.1:=TRUE;
				OP_Regen_Part.Etape.0:=FALSE;
(*étape 1-2*)
ELSIF	OP_Regen_Part.Etape.1
		THEN
				OP_Regen_Part.Etape.2:=TRUE;
				OP_Regen_Part.Etape.1:=FALSE;
(*étape 2-3*)
ELSIF 	OP_Regen_Part.Etape.2
		AND (OP_Isolement.OK
		OR (OP_Pompage_Prim.Etape.0 AND OP_Pompage_Proc.Etape.0 OR OP_Pompage_Sec.Etape.0 OR OP_Purge.Etape.0))
		THEN
				OP_Regen_Part.Etape.3:=TRUE;
				OP_Regen_Part.Etape.2:=FALSE;
(*étape 3-4*)
ELSIF	OP_Regen_Part.Etape.3 AND PS11.STATE_Regen
		THEN
				OP_Regen_Part.Etape.4:=TRUE;
				OP_Regen_Part.Etape.3:=FALSE;
(*étape 4-5*)
ELSIF	OP_Regen_Part.Etape.4
		AND IN_Temp_Etage1 > 300
		THEN
				OP_Regen_Part.Etape.5:=TRUE;
				OP_Regen_Part.Etape.4:=FALSE;
(*étape 5-6*)
ELSIF	OP_Regen_Part.Etape.5
		AND (IN_Temp_Etage1 < PRM_Temp_Post_Purge
			OR TIMER_Post_Purge.Q )
		THEN
				OP_Regen_Part.Etape.6:=TRUE;
				OP_Regen_Part.Etape.5:=FALSE;
(*étape 6-0*)
ELSIF	OP_Regen_Part.Etape.6
		AND TIMER_etape6_regen.Q
		THEN
				OP_Regen_Part.Etape.0:=TRUE;
				OP_Regen_Part.Etape.6:=FALSE;
END_IF;

(*cloture du traitement de l'opération*)
OP_Regen_Part.POST();
END_ACTION

ACTION ACT_TEST_RP:
(*OPERATION TEST REMONTEE PRESSION*)

OP_TEST_RP(
	CTRL_PLC:= CTRL_PLC,
	RESET:= RESET,
	MANUAL:=MANUAL ,
	ENABLE_INT := OP_Pompage_Sec.OK AND OP_Purge.AR AND OP_Regen.AR AND OP_Regen_Part.AR,
	RESTART_ENABLE_IF_OK:=TRUE ,
	N_STEP_OP_OK:= 8,
	N_STEP_OP_NOK:=0 );

(*appel de l'action de préparation de l'opération*)
OP_TEST_RP.PRL();

(*GRAFCET*)
(* initialisation du grafcet*)
IF 		OP_TEST_RP.ETAPE = 0
		THEN
				OP_TEST_RP.ETAPE.0 := TRUE;
(*repositionnement sur étape 0*)
ELSIF 	RESET OR MANUAL OR (OP_Isolement.Etape.1 AND NOT OP_Test_RP.Etape.3)
			OR (OP_Pompage_Sec.Etape.1 AND OP_Test_RP.Etape.3) OR CO_Stop_Test_RP
			OR OP_Arret_Pompes.Etape.1 OR OP_Isolement.ON_AUTO_EXT OR OP_Isolement.ON_AUTO_INT
		THEN
				OP_TEST_RP.ETAPE := 0;
				OP_TEST_RP.ETAPE.0:=TRUE;
(*étape 0-1*)
ELSIF 	OP_TEST_RP.ETAPE.0 AND OP_TEST_RP.MARCHE_OP
		THEN
				OP_TEST_RP.ETAPE.1:=TRUE;
				OP_TEST_RP.ETAPE.0:=FALSE;
(*étape 1-2*)
ELSIF 	OP_TEST_RP.ETAPE.1
		THEN
				OP_TEST_RP.ETAPE.2:=TRUE;
				OP_TEST_RP.ETAPE.1:=FALSE;
(*étape 2-3*)
ELSIF 	OP_TEST_RP.ETAPE.2
		AND OP_Pompage_Sec.ok AND TH_Test_RP
		THEN
				OP_TEST_RP.ETAPE.3:=TRUE;
				OP_TEST_RP.ETAPE.2:=FALSE;
(*étape 3-4*)
ELSIF 	OP_TEST_RP.ETAPE.3
		AND OP_Isolement.OK
		THEN
				OP_TEST_RP.ETAPE.4:=TRUE;
				OP_TEST_RP.ETAPE.3:=FALSE;
(*étape 4-5*)
ELSIF 	OP_TEST_RP.ETAPE.4
		AND TIMER_attente_test.Q
		THEN
				OP_TEST_RP.ETAPE.5:=TRUE;
				OP_TEST_RP.ETAPE.4:=FALSE;
(*étape 5-6*)
ELSIF 	OP_TEST_RP.ETAPE.5
		THEN
				OP_TEST_RP.ETAPE.6:=TRUE;
				OP_TEST_RP.ETAPE.5:=FALSE;
(*étape 6-7*)
ELSIF 	OP_TEST_RP.ETAPE.6
		THEN
				OP_TEST_RP.ETAPE.7:=TRUE;
				OP_TEST_RP.ETAPE.6:=FALSE;
(*étape 7-8*)
ELSIF 	OP_TEST_RP.ETAPE.7
		AND OP_Pompage_Sec.OK
		THEN
				OP_TEST_RP.ETAPE.8:=TRUE;
				OP_TEST_RP.ETAPE.7:=FALSE;
(*étape 8-1*)
ELSIF 	OP_TEST_RP.ETAPE.8 AND OP_TEST_RP.MARCHE_OP
		THEN
				OP_TEST_RP.ETAPE.1:=TRUE;
				OP_TEST_RP.ETAPE.8:=FALSE;
END_IF
(*cloture du traitement de l'opération*)
OP_TEST_RP.POST();
CO_Stop_Test_RP	:=	FALSE;
END_ACTION

ACTION ACT_VENTILATION:
(*OPERATION VENTILATION*)


(*initialisation de l'opération*)
OP_Ventilation(
	CTRL_PLC:= CTRL_PLC,
	RESET:= RESET,
	ENABLE_INT:=OP_Purge.Etape.0,
	MANUAL:= MANUAL,
	ON_AUTO_INT:= FALSE ,
	RESTART_ENABLE_IF_OK:= FALSE,
	N_STEP_OP_OK:= 8,
	N_STEP_OP_NOK:=0);

(*appel de l'action de préparation de l'opération*)
OP_Ventilation.PRL();


(*GRAFCET*)
(* initialisation du grafcet*)
IF 		OP_Ventilation.Etape = 0
		THEN
				OP_Ventilation.Etape.0:= TRUE;
(*repositionnement sur étape 0*)
ELSIF	MANUAL OR RESET OR (OP_isolement.Etape.1 AND NOT  OP_ventilation.Etape.1)
		OR OP_Pompage_sec.Etape.1 OR Op_Pompage_Prim.Etape.1
		OR OP_Pompage_Proc.Etape.1 OR OP_Purge.Etape.1
		THEN
				OP_Ventilation.Etape := 0;
				OP_Ventilation.Etape.0:=TRUE;
(*étape 0-1*)
ELSIF 	OP_Ventilation.Etape.0
		 AND (OP_Ventilation.Marche_OP OR OP_Purge.Etape.4)
		THEN
				OP_Ventilation.Etape.1:=TRUE;
				OP_Ventilation.Etape.0:=FALSE;
(*étape 1-9*)
ELSIF	OP_Ventilation.Etape.1
		AND OP_isolement.OK THEN
				OP_Ventilation.Etape.9:=TRUE;
				OP_Ventilation.Etape.1:=FALSE;
(*étape 9-2*)
ELSIF	OP_Ventilation.Etape.9
		AND OP_isolement.Etape.0 THEN
				OP_Ventilation.Etape.2:=TRUE;
				OP_Ventilation.Etape.9:=FALSE;
(*étape 2-3*)
ELSIF 	OP_Ventilation.Etape.2 AND  I_Prep_Ventil_Ok  THEN
				OP_Ventilation.Etape.3:=TRUE;
				OP_Ventilation.Etape.2:=FALSE;
(*étape 3-4*)
ELSIF	OP_Ventilation.Etape.3
		AND  I_Stop_Mesure_OK   THEN
				OP_Ventilation.Etape.4:=TRUE;
				OP_Ventilation.Etape.3:=FALSE;
(*étape 4-5*)
ELSIF	OP_Ventilation.Etape.4
		THEN
				OP_Ventilation.Etape.5:=TRUE;
				OP_Ventilation.Etape.4:=FALSE;
(*étape 5-6*)
ELSIF 	OP_Ventilation.Etape.5
		AND (TH_atm OR I_Fin_Ventil OR NOT IN_FE11T OR NOT IN_FE12T )
		THEN
				OP_Ventilation.Etape.6:=TRUE;
				OP_Ventilation.Etape.5:=FALSE;
(*étape 6-7*)
ELSIF 	OP_Ventilation.Etape.6
		AND (TIMER_SurVentilation_enc.Q OR I_Fin_Ventil OR NOT IN_FE11T OR NOT IN_FE12T)
		THEN
				OP_Ventilation.Etape.7:=TRUE;
				OP_Ventilation.Etape.6:=FALSE;
(*étape 7-8*)
ELSIF 	OP_Ventilation.Etape.7
		AND VH11.STATE_Off THEN
				OP_Ventilation.Etape.8:=TRUE;
				OP_Ventilation.Etape.7:=FALSE;
END_IF;

(*cloture du traitement de l'opération*)
OP_Ventilation.POST();
END_ACTION

ACTION POST:
VAR_Reset_Sortie := 	NOT MANUAL AND OP_Arret_Pompes.Etape.0 AND OP_Isolement.Etape.0 AND OP_Marche_Pompes.Etape.0
					AND OP_Pompage_Prim.Etape.0 AND OP_Pompage_Proc.Etape.0 AND OP_Pompage_Sec.Etape.0
					AND OP_Ventilation.Etape.0 AND OP_Purge.Etape.0 AND OP_Regen.Etape.0 AND OP_Regen_Part.Etape.0;




(*****************************************)
(*       pompe primaire PP11             *)
(*****************************************)
IF (OP_MARCHE_POMPES.ETAPE.2 AND CONF_Pompage_interjoint)
	OR OP_Pompage_Prim.Etape.3
	OR PS11.STATE_Regen AND NOT RESET
	THEN
		PP11.CO_On 	:= 	TRUE;
ELSIF RESET OR (VAR_Reset_Sortie AND NOT PS11.STATE_Regen)
    OR (OP_Pompage_Sec.Etape.5 AND PR11.STATE_Off AND NOT CONF_Pompage_interjoint)
	OR (OP_Isolement.Etape.3 AND PR11.STATE_Off AND NOT PS11.STATE_Regen  AND NOT CONF_Pompage_interjoint)
	OR OP_Arret_Pompes.Etape.4 AND PR11.STATE_Off AND VP11.STATE_Off
	THEN
		PP11.CO_On	:= 	FALSE;
END_IF;

(*****************************************)
(*       pompe primaire PR11             *)
(*****************************************)
TIMER_Arret_Roots.IN := (OP_Pompage_Sec.OK
						OR (OP_Pompage_Prim.AR AND VP11.STATE_Off AND NOT PS11.STATE_Regen)) AND CONF_Pompage_interjoint;
TIMER_Arret_Roots.PT := T#2M;

TIMER_Arret_Roots();

IF (OP_Pompage_Prim.Etape.3 AND PP11.STATE_On)
	OR (PS11.STATE_Regen AND PP11.STATE_On AND NOT RESET) THEN
		PR11.CO_On 	:= 	TRUE;
ELSIF RESET OR VAR_Reset_Sortie
    OR TIMER_Arret_Roots.Q
	OR OP_Arret_Pompes.Etape.3 
	OR (OP_Isolement.Etape.3 AND NOT PS11.STATE_Regen AND NOT CONF_Pompage_interjoint)
	OR (OP_Pompage_Sec.Etape.5 AND NOT CONF_Pompage_interjoint)
	THEN
		PR11.CO_On	:= 	FALSE;
END_IF;

(*****************************************)
(* 		pompe cryo PS11		   *)
(*****************************************)
IF  OP_Marche_Pompes.Etape.4  THEN
	PS11.CO_On 	:= 	TRUE;
ELSIF RESET  (*OR VAR_Reset_Sortie TODOLN*)  OR OP_Arret_Pompes.Etape.3 THEN
	PS11.CO_On	:= 	FALSE;
	PS11.CO_Regen := FALSE;
END_IF;
IF OP_Regen.Etape.3 OR OP_Regen_Part.Etape.3 THEN
	PS11.CO_Regen	:=	TRUE;
ELSIF OP_Regen.Etape.4 OR OP_Regen_Part.Etape.4 THEN
	PS11.CO_Regen	:=	FALSE;
ELSIF MANUAL THEN
	PS11.CO_On		:=	PS11.VAR_On;
END_IF;

(*****************************************)
(* 		vanne VP11    		   *)
(*****************************************)
IF OP_Pompage_Prim.Etape.4   THEN
		VP11.CO_On 		:= 	TRUE;
ELSIF RESET OR VAR_Reset_Sortie OR OP_Pompage_Sec.Etape.4  OR OP_Isolement.Etape.2 THEN
		VP11.CO_On		:= 	FALSE;
END_IF;


(******************************************)
(*		Vanne  VH11		              *)
(******************************************)
IF   OP_VENTILATION.Etape.5 OR OP_Ventilation.Etape.6 THEN
			VH11.CO_On 	:= 	TRUE;
ELSIF RESET OR  VAR_Reset_Sortie OR OP_Pompage_Prim.Etape.1 OR
	   OP_Pompage_Sec.Etape.2 OR   OP_Isolement.Etape.2 OR OP_Ventilation.Etape.7
	   THEN
			VH11.CO_On	:= 	FALSE;
END_IF;

(******************************************)
(*                  Vanne  VS11                       *)
(******************************************)
IF OP_Pompage_Sec.Etape.6   THEN
		VS11.CO_On 	:= 	TRUE;
		VS11.CO_Lam:=	FALSE;
ELSIF OP_Pompage_Proc.Etape.2  THEN
		VS11.CO_On 	:= 	FALSE;
		VS11.CO_Lam:=	TRUE;
ELSIF VAR_Reset_Sortie OR RESET
	   OR OP_Pompage_Prim.Etape.1   OR OP_Isolement.Etape.2 THEN
		VS11.CO_On	:= 	FALSE;
		VS11.CO_Lam:=	FALSE;
END_IF;


(******************************************)
(*                 Vanne  VINT                        *)
(******************************************)
IF G7_pompage_interjoint.etape.2  THEN
		VINT.CO_On 	:= 	TRUE;
ELSIF VAR_Reset_Sortie OR RESET OR (G7_pompage_interjoint.etape.0 AND NOT MANUAL)
	THEN
		VINT.CO_On	:= 	FALSE;
END_IF;



(***********************************************)
(*                Demande diverse              *)
(***********************************************)

(*demande de préparation avant ventilation*)
RQ_Prep_Ventil_Enc 	:= OP_VENTILATION.Etape.2;

(*Demande d'arrêt de la mesure avant ventilation enceinte*)
RQ_Stop_Mesure_Enc := Op_Ventilation.Etape.3 OR Op_Ventilation.Etape.4 OR Op_Ventilation.Etape.5 ;

(*Tempo de surventilation enceinte*)
TIMER_SurVentilation_Enc	(
					PT:=PRM_Tim_SurVentil_E,
					IN:=OP_VENTILATION.Etape.6 AND TH_Atm
					);

(*Temporisation d'arrêt pompe primaire*)
TIMER_Arret_PP11(
					PT:=PRM_Tim_Arret_PP11,
					IN:=OP_Arret_Pompes.Etape.3,
				);

(*Tempo de purge*)
TIMER_Purge (
					PT:=PRM_Tim_Purge,
					IN:=OP_Purge.Etape.3
					);

(*Compteur d'itération purge*)
IF		OP_Purge.Etape.0 THEN
	VAR_Iter_Purge	:=	0;
ELSIF	OP_Purge.Etape.5 THEN
	VAR_Iter_Purge	:=	VAR_Iter_Purge + 1;
END_IF

(*timer de prep ventil*)
TIM_Prep_ventil.PT := PRM_Tim_Prep_Ventil;
TIM_Prep_ventil.IN := OP_Ventilation.Etape.2;
TIM_Prep_ventil();


(*Tempo de retard à l'ouverture de la vanne interjoint*)
TIMER_pompage_interjoint(
					PT:=T#30s,
					IN:=G7_pompage_interjoint.etape.1
					);


(*timer de post purge en regen partielle*)
TIMER_Post_Purge.PT			:=	PRM_Tim_Post_Purge;
TIMER_Post_Purge.IN			:=	OP_Regen_Part.Etape.5;
TIMER_Post_Purge();

TIMER_etape6_regen.PT		:=	T#500ms;
TIMER_etape6_regen.IN		:=	OP_Regen.Etape.6 OR OP_Regen_Part.Etape.6;
TIMER_etape6_regen();

(***************** test de remontée de pression*************************)
TIMER_attente_test		(
					PT:=PRM_Tim_test,
					IN:=OP_Test_RP.Etape.4
					);
(*Mémorisation des pressions lors du test et calcul de l'indicateur*)
IF FM_etape4.Q THEN
	VAR_Mem_Pression_deb := IN_Pressure_RP;
END_IF;
IF OP_Test_RP.Etape.5 THEN
	VAR_Mem_Pression_fin := IN_Pressure_RP;
END_IF;
(*Indicateur final faisant intervenir le volume ATTENTION : FORMULE MEMO SANS DOUTE FAUSSE*)
IF OP_Test_RP.Etape.6 THEN
	VAR_indicateur_test := (VAR_Mem_Pression_fin - VAR_Mem_Pression_deb) * CONF_volume_enceinte / TIME_TO_REAL(PRM_Tim_Test) * 1000;
END_IF;



(*****************************************************)
(* APPEL DES FONCTIONS COMPOSANTS*)
(*****************************************************)

(*Vanne de pompage primaire enceinte*)
VP11(
	RESET:= RESET,
	MANUAL:= MANUAL,
	EN_On_INT:=  PP11.STATE_On AND PR11.STATE_On AND VH11.STATE_Off AND VS11.STATE_Off AND IN_FE11T AND IN_FE12T AND NOT PS11.STATE_Regen,
	EN_Off_INT:= TRUE
	);

(*Vanne pompage secondaire enceinte*)
VS11(
	RESET:= RESET,
	MANUAL:= MANUAL,
	EN_On_INT:= (PS11.STATE_Ok
				AND VP11.STATE_Off AND VH11.STATE_Off)
				AND TH_RP_Enc,
	EN_Off_INT:= TRUE
	);

(*Vanne ventilation enceinte*)
VH11(
	RESET:= RESET,
	MANUAL:= MANUAL,
	EN_On_INT:= VP11.STATE_Off  AND  VS11.STATE_Off,
	EN_Off_INT:= TRUE
	);

(*Vanne interjoint*)
VINT(
	RESET:= RESET,
	MANUAL:= MANUAL,
	EN_On_INT:= PP11.STATE_On AND NOT PS11.STATE_Regen,
	EN_Off_INT:= TRUE
	);

(*Pompe primaire PP11*)
PP11(
	RESET:= 	RESET,
	MANUAL:= 	MANUAL AND NOT PS11.STATE_Regen,
	EN_On_INT:= TRUE,
	EN_Off_INT:= (PR11.STATE_Off AND VP11.STATE_Off AND NOT PS11.STATE_Regen) OR VAR_Reset_sortie
	);
	
(*Pompe roots PR11*)
PR11(
	RESET:= 	RESET,
	MANUAL:= 	MANUAL,
	EN_On_INT:= PP11.STATE_On,
	EN_Off_INT:= (VP11.STATE_Off AND NOT PS11.STATE_Regen) OR VAR_Reset_sortie
	);

(*Pompe cryo PS11*)
PS11(
	RESET:= RESET,
	MANUAL:= MANUAL,
	EN_On_INT:= TRUE ,
	EN_Off_INT:= VS11.STATE_Off OR VAR_Reset_Sortie,
	EN_Regen_INT:= VS11.STATE_Off
	);


(*******************************************)
(* GESTION DES DEFAUTS 	     *)
(*******************************************)


(*Défaut d'obtention du seuil de basculement en pompage secondaire*)
DEF_PPRIM			(
					Condition:=	(OP_Pompage_Prim.Etape.5 AND OP_Pompage_Sec.Etape.3) AND (DEF_PPRIM.DELAY<>T#0ms)

					);
DEF_TGF				(
					Condition:= 	(OP_Pompage_Prim.Etape.5 OR OP_pompage_prim.Etape.4) AND OP_Pompage_sec.Etape.3
								AND	(DEF_TGF.DELAY<>T#0ms) AND NOT TH_Grosse_Fuite
					);

(*Défaut de remontée de pression dans l'enceinte pendant le pompage secondaire*)
(* validation ok - SP *)
DEF_RP_enc			(
					Condition:=	NOT VS11.STATE_Off AND NOT TH_RP_Enc AND NOT RESET
					);

(*Défaut de ventilation*)
DEF_Vent			(
					Condition:=	(OP_ventilation.Etape.4 OR Op_ventilation.Etape.5 OR op_ventilation.Etape.6) AND (DEF_Vent.DELAY <> T#0ms)
					);
END_ACTION

ACTION PRL:
(*vérification pour empécher la division par 0*)
IF TIME_TO_REAL(PRM_Tim_test) = 0 THEN
	PRM_Tim_test := T#1s;
END_IF
FM_etape4(clk := OP_Test_RP.Etape.4);

	IdXML							:=	'2';
	TagXML							:=	0;

	OP_Marche_Pompes.IdXML			:= 	'1';
	OP_Marche_Pompes.TagXML			:=	1;

	OP_Arret_Pompes.IdXML			:= 	'1';
	OP_Arret_Pompes.TagXML			:= 	2;

	OP_Isolement.IdXML				:= 	'1';
	OP_Isolement.TagXML				:= 	3;

	OP_Ventilation.IdXML			:= 	'1';
	OP_Ventilation.TagXML			:= 	4;

	OP_Pompage_Prim.IdXML			:=	'1';
	OP_Pompage_Prim.TagXML			:=	6;

	OP_Pompage_Sec.IdXML			:=	'1';
	OP_Pompage_Sec.TagXML			:=	5;

	OP_Pompage_Proc.IdXML			:=	'1';
	OP_Pompage_Proc.TagXML			:=	7;

	OP_Purge.IdXML					:=	'1';
	OP_Purge.TagXML					:=	8;

	OP_Regen.IdXML					:=	'1';
	OP_Regen.TagXML					:=	9;

	OP_Test_RP.IdXML				:=	'1';
	OP_Test_RP.TagXML				:=	10;


	DEF_PPrim.IdXML			:= '1';
	DEF_PPrim.TagXML		:= 1;
	DEF_Vent.IdXML			:= '1';
	DEF_Vent.TagXML			:= 2;
	DEF_RP_enc.IdXML		:= '1';
	DEF_RP_enc.TagXML		:= 3;
	DEF_TGF.IdXML			:= '1';
	DEF_TGF.TagXML			:= 4;

	PP11.IdXML					:=	'1';
	PP11.TagXML					:=	7;
	
	PR11.IdXML					:=	'1';
	PR11.TagXML					:=	10;

	PS11.IdXML					:=	'1';
	PS11.TagXML					:=	9;

	VP11.IdXML					:=	'1';
	VP11.TagXML					:=	2;
	VP11.DEF_On.IdXML			:=	'3';
	VP11.DEF_On.TagXML			:=	2;
	VP11.DEF_Off.IdXML			:=	'3';
	VP11.DEF_Off.TagXML			:=	4;
	VP11.DEF_Sensor.IdXML		:=	'3';
	VP11.DEF_Sensor.TagXML		:=	13;
	VP11.DEF_On_Imposs.IdXML	:=	'3';
	VP11.DEF_On_Imposs.TagXML	:=	6;
	VP11.DEF_Off_Imposs.IdXML	:=	'3';
	VP11.DEF_Off_Imposs.TagXML	:=	9;
	VP11.DEF_Off_auto.IdXML		:=	'3';
	VP11.DEF_Off_auto.TagXML	:=	11;

	VH11.IdXML					:=	'1';
	VH11.TagXML					:=	4;
	VH11.DEF_On.IdXML			:=	'3';
	VH11.DEF_On.TagXML			:=	2;
	VH11.DEF_Off.IdXML			:=	'3';
	VH11.DEF_Off.TagXML			:=	4;
	VH11.DEF_Sensor.IdXML		:=	'3';
	VH11.DEF_Sensor.TagXML		:=	13;
	VH11.DEF_On_Imposs.IdXML	:=	'3';
	VH11.DEF_On_Imposs.TagXML	:=	6;
	VH11.DEF_Off_Imposs.IdXML	:=	'3';
	VH11.DEF_Off_Imposs.TagXML	:=	9;
	VH11.DEF_Off_auto.IdXML		:=	'3';
	VH11.DEF_Off_auto.TagXML	:=	11;

	VS11.IdXML					:=	'1';
	VS11.TagXML					:=	3;

	VINT.IdXML					:=	'1';
	VINT.TagXML					:=	1;
	VINT.DEF_On.IdXML			:=	'3';
	VINT.DEF_On.TagXML			:=	2;
	VINT.DEF_Off.IdXML			:=	'3';
	VINT.DEF_Off.TagXML			:=	4;
	VINT.DEF_Sensor.IdXML		:=	'3';
	VINT.DEF_Sensor.TagXML		:=	13;
	VINT.DEF_On_Imposs.IdXML	:=	'3';
	VINT.DEF_On_Imposs.TagXML	:=	6;
	VINT.DEF_Off_Imposs.IdXML	:=	'3';
	VINT.DEF_Off_Imposs.TagXML	:=	9;
	VINT.DEF_Off_auto.IdXML		:=	'3';
	VINT.DEF_Off_auto.TagXML	:=	11;


(* Gestion FM et FD régénération*)
FM_REGEN(CLK:=PS11.STATE_Regen);
FD_REGEN(CLK:=PS11.STATE_Regen);
END_ACTION

END_FUNCTION_BLOCK

(* stored: Version 1.1.0.1, ProductVersion 3.1.4024.12
   POU BLOCK_POMP_1E_PCR_PPM_ASS_ETHERCAT: Id {ee7ae957-b402-4700-ab0f-336521f622c9}, SpecialFunc None
   Action ACT_ARRET_POMPES: Id {68597c66-a2a0-40fb-a14f-f64e80d845b4}
   Action ACT_ISOLEMENT: Id {7ff1bd5b-f397-4a38-ab58-2bc41a96e209}
   Action ACT_MARCHE_POMPES: Id {59e04edd-1731-4d9e-81ab-9d0dfb5d4e72}
   Action ACT_POMPAGE_INTERJOINT: Id {4a72685f-d064-4846-a0b7-76d792cb4a63}
   Action ACT_POMPAGE_PRIM: Id {428afd81-72ef-4132-869c-ffe20e55f7ba}
   Action ACT_POMPAGE_PROC: Id {add7c0c1-4150-460f-8873-44da9ae8d09d}
   Action ACT_POMPAGE_SEC: Id {dc00ed62-4d1a-4b70-b3a7-cfc47f27f1d2}
   Action ACT_PURGE: Id {5c7f2e55-f9e4-48b4-a646-948d4dcf2b17}
   Action ACT_REGEN: Id {96f5081d-cf60-45ed-976b-efa75f6f02b4}
   Action ACT_REGEN_PART: Id {c9af2f62-1496-4e21-86db-688f5bffac06}
   Action ACT_TEST_RP: Id {03b0dcc1-7eaa-4e33-8ea3-2e92665f0cc8}
   Action ACT_VENTILATION: Id {54bfd8ab-e798-4540-bd17-a9e4fc13c922}
   Action POST: Id {bb5ce370-cf0b-4199-afee-301ea5f8bbb2}
   Action PRL: Id {f30e021f-99b4-432c-8fd4-6c7fcbcf0446} *)
